// TIA Portal V16 export
// export: Created 2024-05-13T12:47:23.1745312Z, ExportSetting WithDefaults, DisplayName Totally Integrated Automation Portal, DisplayVersion V16 Update 6, DisplayName TIA Portal Version Control Interface, DisplayVersion V16 Update 2, DisplayName TIA Portal Openness, DisplayVersion V16 Update 6, DisplayName TIA Portal Test Suite Advanced, DisplayVersion V16, DisplayName SINAMICS Startdrive Advanced, DisplayVersion V16 Update 5, DisplayName SINAMICS Startdrive G130, G150, S120, S150, SINAMICS MV, S210, DisplayVersion V16 Update 5, DisplayName SINAMICS Startdrive G110M, G120, G120C, G120D, G120P, G115D, DisplayVersion V16 Update 5, DisplayName STEP 7 Professional, DisplayVersion V16 Update 6, DisplayName STEP 7 Safety, DisplayVersion V16, DisplayName WinCC Advanced, DisplayVersion V16 Update 6
TYPE "SCA_labelApplicator_IO_Input"
// stored: IsFailsafeCompliant false
   STRUCT
      Safety_switch : Bool;   // Safety switch
      Up_limit : Bool;   // Up limit
      Down_limit : Bool;   // Down limit
      Area_free_1 : Bool;   // Area free 1
      Area_free_2 : Bool;   // Area free 2
      Roll_sensing_1 : Bool;   // Roll sensing 1
      Roll_sensing_2 : Bool;   // Roll sensing 2
      Brake_fuse : Bool;   // Brake fuse OK
      HS1_spare : Bool;   // Handshake, spare
      HS2_piston_at_home : Bool;   // Handshake, piston at home
      HS3_warning : Bool;   // Handshake, warning
      HS4_fault : Bool;   // Handshake, fault
      Man_up : Bool;   // Manual up switch
      Man_down : Bool;   // Manual down switch
   END_STRUCT;
END_TYPE
